// TIA Portal project "Ejercicio3" (V15.1)

(* hardware
DEVICE "HMI_1"  KTP700 Basic PN
   slot 0: "HMI_1"  KTP700 Basic PN  6AV2 123-2GB03-0AX0  15.1.0.0
   slot 1: "HMI_RT_1"  KTP700 Basic PN  6AV2 123-2GB03-0AX0  15.1.0.0
   slot 5: "HMI_1.IE_CP_1"  PROFINET Interface  15.0.1.0
      slot 1: "Interfaz PROFINET_1"  PROFINET Interface
         slot 1: "Port_1"  Port
DEVICE "S7-1200 station_1"  S7-1200 Station
   slot 0: "Rack_0"  S7-1200 Rack  Rack  V1.0
   slot 1: "PLC_1"  CPU 1215C AC/DC/Rly  6ES7 215-1BG40-0XB0  V4.2
*)

// ===== PLC "PLC_1"  CPU 1215C AC/DC/Rly =====

VAR_GLOBAL   // PLC tag table "Tabla de variables estándar"
   "Marcha" AT %M0.0 : Bool;
   "Paro" AT %M0.1 : Bool;
   "Pila de pales en entrada" AT %M0.2 : Bool;
   "Pila de pales en desapilador" AT %M0.3 : Bool;
   "Pale en rodillos de salida" AT %M0.4 : Bool;
   "Cilindro subir pilas pales reposo" AT %M0.5 : Bool;
   "Cilindro subir pilas pales arriba" AT %M0.6 : Bool;
   "Cilindro uña sujetar pila reposo" AT %M0.7 : Bool;
   "Cilindro uña sujetar pila extendida" AT %M1.0 : Bool;
   "Freno pila recogido" AT %M1.1 : Bool;
   "Freno pila extendido" AT %M1.2 : Bool;
   "Motor rodillos entrada pilas" AT %M10.0 : Bool;
   "Motor rodillos desapilador" AT %M10.1 : Bool;
   "Motor rodillos salida pale" AT %M10.2 : Bool;
   "Cilindro subir pila" AT %M10.3 : Bool;
   "Cilindro uña sujetar pila" AT %M10.4 : Bool;
   "Cilindro freno" AT %M10.5 : Bool;
   "Permiso  extracción  pale" AT %M2.0 : Bool;
END_VAR

// folder: System blocks/Program resources

DATA_BLOCK "IEC_Timer_0_DB"   // DB1
{ S7_Optimized_Access := 'TRUE' }
AUTHOR : Simatic
FAMILY : IEC
NAME : IEC_TMR
VERSION : 1.0
// stored: InstanceOfName IEC_TIMER
"IEC_TIMER"
BEGIN
END_DATA_BLOCK

DATA_BLOCK "IEC_Timer_0_DB_1"   // DB2
{ S7_Optimized_Access := 'TRUE' }
AUTHOR : Simatic
FAMILY : IEC
NAME : IEC_TMR
VERSION : 1.0
// stored: InstanceOfName IEC_TIMER
"IEC_TIMER"
BEGIN
END_DATA_BLOCK

DATA_BLOCK "IEC_Timer_0_DB_2"   // DB3
{ S7_Optimized_Access := 'TRUE' }
AUTHOR : Simatic
FAMILY : IEC
NAME : IEC_TMR
VERSION : 1.0
// stored: InstanceOfName IEC_TIMER
"IEC_TIMER"
BEGIN
END_DATA_BLOCK

// folder: (top level)

ORGANIZATION_BLOCK "Main"   // OB1, LAD, ProgramCycle
TITLE = "Main Program Sweep (Cycle)"
{ S7_Optimized_Access := 'TRUE' }
VERSION : 0.1
   VAR_INPUT
      Initial_Call : Bool;   // Initial call of this OB
      Remanence : Bool;   // =True, if remanent data are available
   END_VAR
BEGIN

REGION Network 1
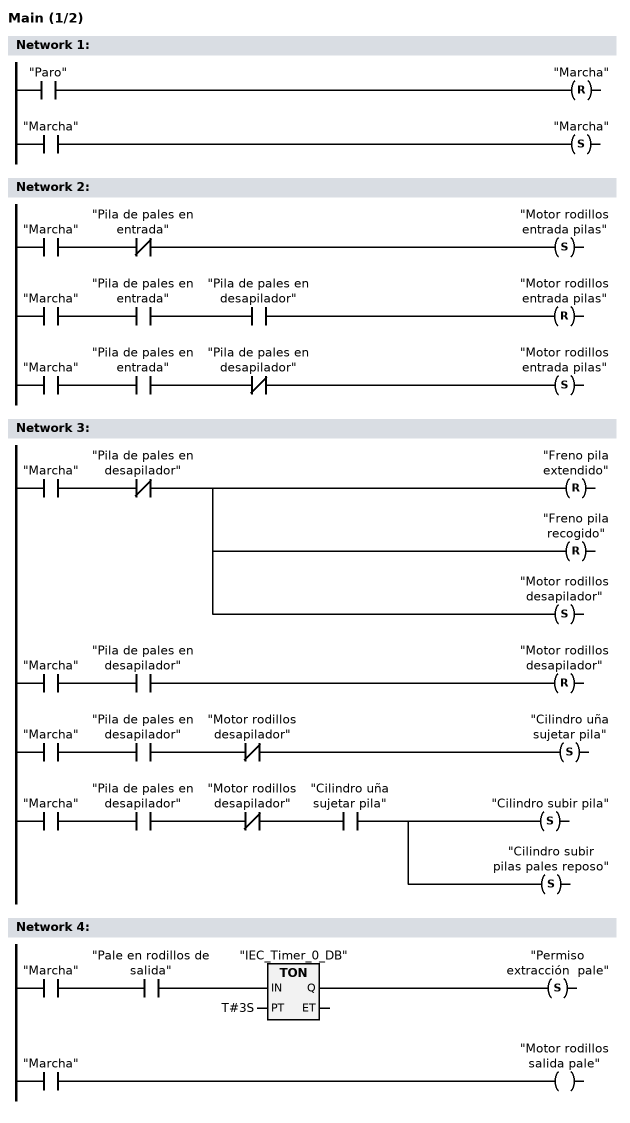
   RUNG wire#powerrail
      Contact( "Paro" )
      R_Coil( "Marcha" )
   END_RUNG
   RUNG wire#powerrail
      Contact( "Marcha" )
      S_Coil( "Marcha" )
   END_RUNG
   // the same network as SCL:
   IF "Paro" THEN "Marcha" := FALSE; END_IF;
   IF "Marcha" THEN "Marcha" := TRUE; END_IF;
END_REGION

REGION Network 2
   RUNG wire#powerrail
      Contact( "Marcha" )
      I_Contact( "Pila de pales en entrada" )
      S_Coil( "Motor rodillos entrada pilas" )
   END_RUNG
   RUNG wire#powerrail
      Contact( "Marcha" )
      Contact( "Pila de pales en entrada" )
      Contact( "Pila de pales en desapilador" )
      R_Coil( "Motor rodillos entrada pilas" )
   END_RUNG
   RUNG wire#powerrail
      Contact( "Marcha" )
      Contact( "Pila de pales en entrada" )
      I_Contact( "Pila de pales en desapilador" )
      S_Coil( "Motor rodillos entrada pilas" )
   END_RUNG
   // the same network as SCL:
   IF "Marcha" AND NOT "Pila de pales en entrada" THEN "Motor rodillos entrada pilas" := TRUE; END_IF;
   IF "Marcha" AND "Pila de pales en entrada" AND "Pila de pales en desapilador" THEN
       "Motor rodillos entrada pilas" := FALSE;
   END_IF;
   IF "Marcha" AND "Pila de pales en entrada" AND NOT "Pila de pales en desapilador" THEN
       "Motor rodillos entrada pilas" := TRUE;
   END_IF;
END_REGION

REGION Network 3
   RUNG wire#powerrail
      Contact( "Marcha" )
      I_Contact( "Pila de pales en desapilador" )
      wire#w1
      R_Coil( "Freno pila extendido" )
   END_RUNG
   RUNG wire#w1
      R_Coil( "Freno pila recogido" )
   END_RUNG
   RUNG wire#w1
      S_Coil( "Motor rodillos desapilador" )
   END_RUNG
   RUNG wire#powerrail
      Contact( "Marcha" )
      Contact( "Pila de pales en desapilador" )
      R_Coil( "Motor rodillos desapilador" )
   END_RUNG
   RUNG wire#powerrail
      Contact( "Marcha" )
      Contact( "Pila de pales en desapilador" )
      I_Contact( "Motor rodillos desapilador" )
      S_Coil( "Cilindro uña sujetar pila" )
   END_RUNG
   RUNG wire#powerrail
      Contact( "Marcha" )
      Contact( "Pila de pales en desapilador" )
      I_Contact( "Motor rodillos desapilador" )
      Contact( "Cilindro uña sujetar pila" )
      wire#w2
      S_Coil( "Cilindro subir pila" )
   END_RUNG
   RUNG wire#w2
      S_Coil( "Cilindro subir pilas pales reposo" )
   END_RUNG
   // the same network as SCL:
   IF "Marcha" AND NOT "Pila de pales en desapilador" THEN
       "Freno pila extendido" := FALSE;
       "Freno pila recogido" := FALSE;
       "Motor rodillos desapilador" := TRUE;
   END_IF;
   IF "Marcha" AND "Pila de pales en desapilador" THEN "Motor rodillos desapilador" := FALSE; END_IF;
   IF "Marcha" AND "Pila de pales en desapilador" AND NOT "Motor rodillos desapilador" THEN
       "Cilindro uña sujetar pila" := TRUE;
   END_IF;
   IF "Marcha" AND "Pila de pales en desapilador" AND NOT "Motor rodillos desapilador" AND "Cilindro uña sujetar pila" THEN
       "Cilindro subir pila" := TRUE;
       "Cilindro subir pilas pales reposo" := TRUE;
   END_IF;
END_REGION

REGION Network 4
   "IEC_Timer_0_DB".TON(IN := "Marcha" AND "Pale en rodillos de salida", PT := T#3S);
   IF "IEC_Timer_0_DB".Q THEN "Permiso  extracción  pale" := TRUE; END_IF;
   "Motor rodillos salida pale" := "Marcha";
END_REGION

REGION Network 5
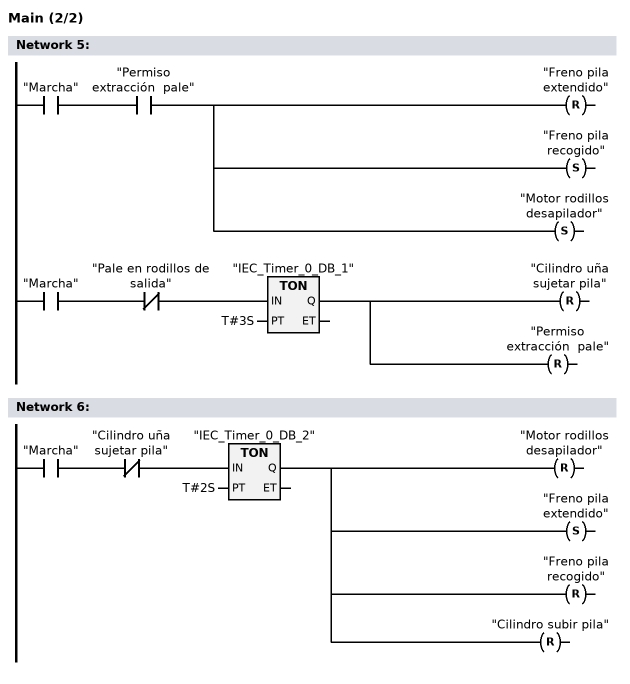
   IF "Marcha" AND "Permiso  extracción  pale" THEN
       "Freno pila extendido" := FALSE;
       "Freno pila recogido" := TRUE;
       "Motor rodillos desapilador" := TRUE;
   END_IF;
   "IEC_Timer_0_DB_1".TON(IN := "Marcha" AND NOT "Pale en rodillos de salida", PT := T#3S);
   IF "IEC_Timer_0_DB_1".Q THEN
       "Cilindro uña sujetar pila" := FALSE;
       "Permiso  extracción  pale" := FALSE;
   END_IF;
END_REGION

REGION Network 6
   "IEC_Timer_0_DB_2".TON(IN := "Marcha" AND NOT "Cilindro uña sujetar pila", PT := T#2S);
   IF "IEC_Timer_0_DB_2".Q THEN
       "Motor rodillos desapilador" := FALSE;
       "Freno pila extendido" := TRUE;
       "Freno pila recogido" := FALSE;
       "Cilindro subir pila" := FALSE;
   END_IF;
END_REGION
END_ORGANIZATION_BLOCK

(* ===== HMI "HMI_RT_1" =====
system functions are stored by id; their names below are inferred from use
connection "HMI_Conexión_1": ETHERNET, SMART_S7_1200_OMS

HMI tags "Tabla de variables estándar"
   "Número_imagen_variable" : UInt, internal
   "Pila de pales en entrada" : Bool = PLC "Pila de pales en entrada" AT %M0.2, 1 s
   "Pila de pales en desapilador" : Bool = PLC "Pila de pales en desapilador" AT %M0.3, 1 s
   "Pale en rodillos de salida" : Bool = PLC "Pale en rodillos de salida" AT %M0.4, 1 s
   "Cilindro subir pilas pales reposo" : Bool = PLC "Cilindro subir pilas pales reposo" AT %M0.5, 1 s
   "Cilindro subir pilas pales arriba" : Bool = PLC "Cilindro subir pilas pales arriba" AT %M0.6, 1 s
   "Cilindro uña sujetar pila reposo" : Bool = PLC "Cilindro uña sujetar pila reposo" AT %M0.7, 1 s
   "Cilindro uña sujetar pila extendida" : Bool = PLC "Cilindro uña sujetar pila extendida" AT %M1.0, 1 s
   "Freno pila recogido" : Bool = PLC "Freno pila recogido" AT %M1.1, 1 s
   "Freno pila extendido" : Bool = PLC "Freno pila extendido" AT %M1.2, 1 s

text list "Nombre_imagen_lista_texto": 1 'Imagen raíz'

Template "Plantilla_1" 800x480
   Button "Salir" at 714,429 size 71x50; TextOff 'Salir'; PictureOff "ExitRuntime_KTP700_Basic_PN_TR"; PictureOn "ExitRuntime_KTP700_Basic_PN_TR"
      on Release: StopRuntime(0)
   Button "Template_Button" at 614,429 size 71x50; TextOff 'Text'
   Button "Template_Button_1" at 514,429 size 71x50; TextOff 'Text'
   Button "Template_Button_2" at 414,429 size 71x50; TextOff 'Text'
   Button "Template_Button_3" at 314,429 size 71x50; TextOff 'Text'
   Button "Template_Button_4" at 214,429 size 71x50; TextOff 'Text'
   Button "Template_Button_5" at 114,429 size 71x50; TextOff 'Text'
   Button "Imagen inicial" at 14,429 size 71x50; TextOff 'Imagen inicial'; PictureOff "NavigateHome_KTP700_Basic_PN_TR"; PictureOn "NavigateHome_KTP700_Basic_PN_TR"
      on Release: ActivateScreen("Imagen raíz", 0)
   SymbolicIOField "Imagen_campo_ES_simbólico" at 93,9 size 600x33; TextOff '0'; TextOn '1'; TextList "Nombre_imagen_lista_texto"
      ProcessValue <- "Número_imagen_variable"
      on Change: ActivateScreenByNumber("Número_imagen_variable", 0)
   DateTimeField "HmiScreenItemData" at 695,25 size 105x25
   DateTimeField "HmiScreenItemData_1" at 695,0 size 105x25
   GraphicView "Logotipo" at 0,0 size 91x51; Picture "Logotipo de HMI_1"

screen "Imagen raíz" 800x480, template "Plantilla_1"
   on GenerateScreen: SetTag("Número_imagen_variable", 1)
   Switch "Interruptor_1" at 59,115 size 96x32; CaptionText 'Switch'; TextOff 'OFF'; TextOn 'ON'
   Button "Botón_1" at 170,103 size 150x56; TextOff 'Boton Paro'
   TextField "Campo de texto_4" at 401,70 size 168x23; Text 'Estado freno M2-M3'
   TextField "Campo de texto_5" at 401,138 size 236x23; Text 'Estado cilindro Arriba/abajo'
   Switch "Interruptor_2" at 53,214 size 64x32; CaptionText 'Switch'; TextOff 'OFF'; TextOn 'ON'
      ProcessValue <- "Pila de pales en entrada"
   Switch "Interruptor_3" at 214,214 size 64x32; TextOn 'ON'; CaptionText 'Switch'; TextOff 'OFF'
      ProcessValue <- "Pila de pales en desapilador"
   Switch "Interruptor_4" at 450,214 size 64x32; TextOn 'ON'; CaptionText 'Switch'; TextOff 'OFF'
      ProcessValue <- "Pale en rodillos de salida"
   Switch "Interruptor_5" at 652,214 size 64x32; TextOn 'ON'; CaptionText 'Switch'; TextOff 'OFF'
      ProcessValue <- "Cilindro subir pilas pales reposo"
   Switch "Interruptor_6" at 53,315 size 64x32; TextOn 'ON'; CaptionText 'Switch'; TextOff 'OFF'
      ProcessValue <- "Cilindro subir pilas pales arriba"
   Switch "Interruptor_7" at 212,315 size 64x32; TextOn 'ON'; CaptionText 'Switch'; TextOff 'OFF'
      ProcessValue <- "Cilindro uña sujetar pila reposo"
   Switch "Interruptor_8" at 652,315 size 64x32; TextOn 'ON'; CaptionText 'Switch'; TextOff 'OFF'
      ProcessValue <- "Cilindro uña sujetar pila extendida"
   Switch "Interruptor_9" at 53,388 size 64x32; TextOn 'ON'; CaptionText 'Switch'; TextOff 'OFF'
      ProcessValue <- "Freno pila recogido"
   Switch "Interruptor_10" at 214,388 size 64x32; TextOn 'ON'; CaptionText 'Switch'; TextOff 'OFF'
      ProcessValue <- "Freno pila extendido"
   TextField "Campo de texto_1" at 20,186 size 150x23; Text 'Palets en entrada'
   TextField "Campo de texto_2" at 180,186 size 181x23; Text 'Palets en desapilador'
   TextField "Campo de texto_3" at 397,186 size 134x23; Text 'Palets en salida'
   TextField "Campo de texto_6" at 601,180 size 190x23; Text 'Subir pila pales reposo'
   TextField "Campo de texto_7" at 5,287 size 184x23; Text 'Subir pila pales arriba'
   TextField "Campo de texto_8" at 199,287 size 261x23; Text 'Cilindro uña sujetar pila reposo'
   TextField "Campo de texto_9" at 512,287 size 288x23; Text 'Cilindro uña sujetar pila extendida'
   TextField "Campo de texto_10" at 1,365 size 161x23; Text 'Freno pila recogido'
   TextField "Campo de texto_11" at 184,365 size 173x23; Text 'Freno pila extendido'
*)